// TIA Portal V20 program export: 1 tag tables, 3 data types, 5 data blocks, 3 code blocks (in call order from the OBs), 0 instance data blocks

VAR_GLOBAL   // PLC tag table "Gate1"
   Prox1 AT %I0.0 : Bool;   // Stato sensore prossimità cancello 1 (Aperto -> False)
   Prox2 AT %I0.1 : Bool;   // Stato sensore prossimità cancello 2 (Aperto -> False)
   Prox3 AT %I0.2 : Bool;   // Stato sensore prossimità cancello 3 (Aperto -> False)
END_VAR

TYPE "MaxMin"
   STRUCT
      Min : Real;
      Max : Real;
   END_STRUCT;
END_TYPE

TYPE "Position"
   STRUCT
      LinAxis : Struct   // Assi lineari
         X : Real;
         Y : Real;
         Z : Real;
      END_STRUCT;
      AngAxis : Struct   // Assi angolari
         "B" : Real;
         C : Real;
      END_STRUCT;
   END_STRUCT;
END_TYPE

TYPE "Stroke"
   STRUCT
      LinaAxis : Struct
         X : "MaxMin";
         Y : "MaxMin";
         Z { S7_SetPoint := 'True'} : "MaxMin";
      END_STRUCT;
      AngAxis : Struct
         "B" : "MaxMin";
         C : "MaxMin";
      END_STRUCT;
   END_STRUCT;
END_TYPE

DATA_BLOCK "InputData"   // DB1
TITLE = Dati in ingresso
{ S7_Optimized_Access := 'TRUE' }
AUTHOR : Nicola
// DB che raccogie di dati letti dai sensori in campo
// stored: MemoryReserve 100
   VAR
      Gt1IsClosed : Bool;   // Cancello 1 chiuso (False -> Aperto)
      Gt2IsClosed : Bool;   // Cancello 2 chiuso (False -> Aperto)
      Gt3IsClosed : Bool;   // Cancello 3 chiuso (False -> Aperto)
   END_VAR
BEGIN
END_DATA_BLOCK

DATA_BLOCK "CurrGlob"   // DB3
TITLE = Dati di posizione in coordinate assolute
{ S7_Optimized_Access := 'TRUE' }
// Ottiene la passizione assoluta degli assi
// stored: MemoryReserve 100
   VAR
      Pos : "Position";
   END_VAR
BEGIN
END_DATA_BLOCK

DATA_BLOCK "CurrStroke"   // DB5
TITLE = Valori delle corse macchina attuali
{ S7_Optimized_Access := 'TRUE' }
// Sava i dati di valore Minimo e Massimo per gli assi correnti
// stored: MemoryReserve 100
   VAR
      Str : "Stroke";
   END_VAR
BEGIN
END_DATA_BLOCK

DATA_BLOCK "TargetGlob"   // DB4
TITLE = Setta il punto di arrivo proìevisto
{ S7_Optimized_Access := 'TRUE' }
AUTHOR : Nicola
// Imposta la posizione in coordiate assolute da raggiungere
// stored: MemoryReserve 100
   VAR
      Pos : "Position";
   END_VAR
BEGIN
END_DATA_BLOCK

DATA_BLOCK "Appo"   // DB2
TITLE = Variabili di appoggio
{ S7_Optimized_Access := 'TRUE' }
// Per spostare dati nel sw in modo facile
// stored: MemoryReserve 100
   VAR
      Gt1St : Byte;
   END_VAR
BEGIN
END_DATA_BLOCK

ORGANIZATION_BLOCK "Main"   // OB1, LAD, ProgramCycle
TITLE = "Main Program Sweep (Cycle)"
{ S7_Optimized_Access := 'TRUE' }
// stored: SetENOAutomatically false
   VAR_INPUT
      Initial_Call : Bool;   // Initial call of this OB
      Remanence : Bool;   // =True, if remanent data are available
   END_VAR
   VAR_TEMP   // added for the SCL form of the ladder/FBD networks
      _w1 : Bool;
   END_VAR
BEGIN

REGION Network 1
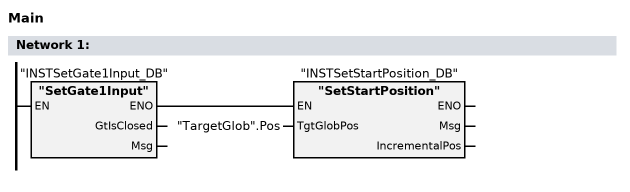
   RUNG wire#powerrail
      "INSTSetGate1Input_DB"(GtIsClosed =>, Msg =>)
      "INSTSetStartPosition_DB"(TgtGlobPos := "TargetGlob".Pos, Msg =>, IncrementalPos =>)
   END_RUNG
   // the same network as SCL:
   "INSTSetGate1Input_DB"(ENO => #_w1);   // "SetGate1Input"
   IF #_w1 THEN
       "INSTSetStartPosition_DB"(TgtGlobPos := "TargetGlob".Pos);   // "SetStartPosition"
   END_IF;
END_REGION
END_ORGANIZATION_BLOCK

FUNCTION_BLOCK "SetGate1Input"
TITLE = Imposta stato delle variabili relative alle porte
{ S7_Optimized_Access := 'TRUE' }
AUTHOR : Nicola
VERSION : 0.1
//Carico lo stato delle variabili porte
   VAR_INPUT 
      Ind : Int;
   END_VAR

   VAR_OUTPUT 
      GtIsClosed : Bool;
      Msg : String := '';
   END_VAR


BEGIN
	// Carico i dati del letti dalle TAG nel DB 
	"InputData".Gt1IsClosed := "Prox1";
	"InputData".Gt2IsClosed := "Prox2";
	"InputData".Gt3IsClosed := "Prox3";
	#Msg := 'Waiting Status';
	// Stato porta 1 - Messaggio per lettura semplificata
	IF "InputData".Gt1IsClosed THEN
	    #Msg := 'Porta 1 chiusa';
	    "Appo".Gt1St.%X0 := 1;
	ELSE
	    #Msg := 'Porta 1 aperta';
	    "Appo".Gt1St.%X0 := 0;
	END_IF;
	// Stato porta 2
	IF "InputData".Gt2IsClosed THEN
	    #Msg := CONCAT(IN1 := #Msg, IN2 := ' - Porta 2 chiusa');
	    "Appo".Gt1St.%X1 := 1;
	ELSE
	    #Msg := CONCAT(IN1 := #Msg, IN2 := ' - Porta 2 aperta');
	    "Appo".Gt1St.%X1 := 0;
	END_IF;
	// Stato porta 3
	IF "InputData".Gt3IsClosed THEN
	    #Msg := CONCAT(IN1 := #Msg, IN2 := ' - Porta 3 chiusa');
	    "Appo".Gt1St.%X2 := 1;
	ELSE
	    #Msg := CONCAT(IN1 := #Msg, IN2 := ' - Porta 3 aperta');
	    //"Appo".Gt1St.%X2 := 0;
	END_IF;
	
	// Cumulativo
	#GtIsClosed := "InputData".Gt1IsClosed AND "InputData".Gt2IsClosed AND "InputData".Gt3IsClosed;
	
	// Salvo nel vettore nella posizione specificata il valore opposto a quello correntemente salvato
	"Appo".VtInt[#Ind] := NOT "Appo".VtInt[#Ind];
	
END_FUNCTION_BLOCK

FUNCTION_BLOCK "SetStartPosition"
TITLE = Prepara i dati per il posizionamento
{ S7_Optimized_Access := 'TRUE' }
AUTHOR : Nicola
VERSION : 0.1
//Imposto le posizioni che devono essere raggiunte per poter iniziare una lavorazione
   VAR_INPUT 
      TgtGlobPos : "Position";   // Valore di posizione targe i coordinate globali
   END_VAR

   VAR_OUTPUT 
      Msg { ExternalAccessible := 'False'; ExternalVisible := 'False'; ExternalWritable := 'False'} : String;
      IncrementalPos : "Position";
   END_VAR

   VAR 
      Ok : Bool;
   END_VAR


BEGIN
	REGION "Verifica posizione nei limiti macchina"
	    
	    // Verifcìico asse X
	    IF #TgtGlobPos.LinAxis.X < "CurrStroke".Str.LinaAxis.X.Max AND #TgtGlobPos.LinAxis.X > "CurrStroke".Str.LinaAxis.X.Min THEN
	        #Ok := TRUE;
	    END_IF;
	    
	    // Verifcìico asse Y
	    IF #TgtGlobPos.LinAxis.Y < "CurrStroke".Str.LinaAxis.Y.Max AND #TgtGlobPos.LinAxis.Y > "CurrStroke".Str.LinaAxis.Y.Min THEN
	        #Ok := TRUE;
	    END_IF;
	    
	    // Verifcìico asse Z
	    IF #TgtGlobPos.LinAxis.Z < "CurrStroke".Str.LinaAxis.Z.Max AND #TgtGlobPos.LinAxis.Z > "CurrStroke".Str.LinaAxis.Z.Min THEN
	        #Ok := TRUE;
	    END_IF;
	    
	END_REGION
	
	REGION "Calcolo valore incrementale"
	    
	    // Se la verifica dei limiti corsa è corretta allora calcolo il valore incrementale
	    IF #Ok THEN
	        #IncrementalPos.LinAxis.X := #TgtGlobPos.LinAxis.X - "CurrGlob".Pos.LinAxis.X;
	        #IncrementalPos.LinAxis.Y := #TgtGlobPos.LinAxis.Y - "CurrGlob".Pos.LinAxis.Y;
	        #IncrementalPos.LinAxis.Z := #TgtGlobPos.LinAxis.X - "CurrGlob".Pos.LinAxis.Z;
	    END_IF;
	        
	END_REGION
	
END_FUNCTION_BLOCK
